(* CODESYS project filling_station_1309_Final.ecp

Project tree, tasks and I/O mapping:
  GenericDummyMasterDevice : Generic Master, WAGO, order no. None, version 1.0.0.0
  PFC200_CS_2ETH_RS : 750-8202 PFC200 2ETH RS, WAGO, order no. 0750-8202, version 1.4.1.22
    application Application
      libraries: ; Util, * (System); VisuDialogs, * (System)
      task PLC_Task (cyclic, interval t#10ms, priority 14) calls PLC_PRG
      task Visu_Task (cyclic, interval t#10ms, priority 14) calls VISU_PRG
      function CONVERT_PRESSURE_TO_LEVEL [ST]
      visualisation Visualization
      function READ_PRESSURE [ST]
      global variables GVL
      function XOR_MANUAL_AUTOMATIC_VALVE_CONTROL [ST]
      function READ_VALVE_POSITION [ST]
      function AVOID_SIMULT_VALVE_OPEN_AND_CLOSE [ST]
      program PLC_PRG [FBD]
      image pool ImagePool
      visualisation Visualization_1
      function ASSIGN_OUTPUTS [ST]
      function ACTUATOR [ST]
      function Manual_Control [FBD]
    DeviceAdapter
    Kbus : Kbus, WAGO, version 1.3.0.0
        unmapped channels: K-BUS diagnostics
      _8_DO_Generic : 075x-8DO, WAGO, order no. 075x-8DO, version 0.0.0.11
          settings: K-BUS Module slot index = 1
          output vbOpenSamsonValve : BOOL  // _OUT._OUT
          output vbCloseSamsonValve : BOOL  // _OUT._OUT
          output vbOpenDrainValveBelowWaterColumn : BOOL  // _OUT._OUT
          output vbSwitchOnPump : BOOL  // _OUT._OUT
          unmapped channels: _OUT
        DeviceAdapter
      _4_AI_0_10V_DC_s_e : 0750-0459, WAGO, order no. 0750-0459, version 0.0.0.11
          settings: K-BUS Module slot index = 2
          input  vwRawValvePosition : WORD  // _IW 1
          unmapped channels: _IW 2, _IW 3, _IW 4
        DeviceAdapter
      _2_AI_4_20mA_Diff_Measurement_Input : 0750-0492, WAGO, order no. 0750-0492, version 0.0.0.7
          settings: K-BUS Module slot index = 3
          input  vwRawPressure : WORD  // _IW 1
          unmapped channels: _IW 2
        DeviceAdapter
    MODBUS
      MODBUS : MODBUS, WAGO, order no. n/a, version 1.1.1.13
    Serial
      COM1 : COM1, WAGO, version 0.0.0.19
  e_DISPLAY_7300T_WP_10_1_1280x800_PIO1 : 0762-3003 e!DISPLAY 7300T - WP 10.1, WAGO, order no. 0762-3003, version 0.0.0.3
    DeviceAdapter
  libraries: WagoVisuIcons, 1.0.0.7 (WAGO)
  text list GlobalTextList
  5ce3da45-db07-42e7-a21c-a00fff4ed8f6|C:\Users\Alexander Wilms\Documents\Ausbildung\Hochschule Darmstadt\Master Electrical Engineering\1. Semester\Team Project\team-project\40_Implementation\hydraulics-schematic-simplified.png
  5ce3da45-db07-42e7-a21c-a00fff4ed8f6|C:\Users\Alexander Wilms\Documents\Ausbildung\Hochschule Darmstadt\Master Electrical Engineering\1. Semester\Team Project\team-project\30_Architecture\hydraulics-schematic-simplified.png
*)

// PFC200_CS_2ETH_RS/Application/GVL
VAR_GLOBAL
	vrWaterLevel:REAL;
	vrgrWaterLevel:ARRAY[1..16] OF REAL;
	vrStandardGravity:REAL:=9.81;
	viDensityWater:INT:=1000;
	vrValvePosition:REAL;
	vrValvePositionPercentage:REAL;
	vrValvePositionDesired:REAL;
	viPumpPowerPercentage:INT;
	vbManualValveControl:BOOL:=TRUE;
	vbAutomaticValveControl:BOOL:=FALSE;
	vbPreviousValveControl:STRING:='MANUAL';
	vbPreviousSamsonValveDirection:STRING:='STOP';
	vbStopSamsonValve:BOOL:=TRUE;
	vbOpenSamsonValveButton:BOOL;
	vbCloseSamsonValveButton:BOOL;
	vbOpenSamsonValveCtrl:BOOL;
	vbCloseSamsonValveCtrl:BOOL;
	vbSwitchOnPumpCtrl:BOOL:=FALSE;
	vbTrash: BOOL;
	vrController_Level_SP:REAL;
	vrController_PV:REAL;
	vbController_Manual_Mode:BOOL:=TRUE;
	vrController_Output:REAL;
	vrController_Output_reversed:REAL;
	Water_Valve_Open: BOOL;
	Water_Valve_Close: BOOL;
	PID_1: PID;
	vbOpenDrainValveBelowWaterColumnCtrl: BOOL;
END_VAR
VAR_GLOBAL RETAIN
	KP: REAL:=0.7;
	TN: REAL:=3;
	TV: REAL:=0;
END_VAR

// PFC200_CS_2ETH_RS/Application/PLC_PRG
PROGRAM PLC_PRG
VAR
	PID_0: PID;
	TRASH: BOOL;
END_VAR

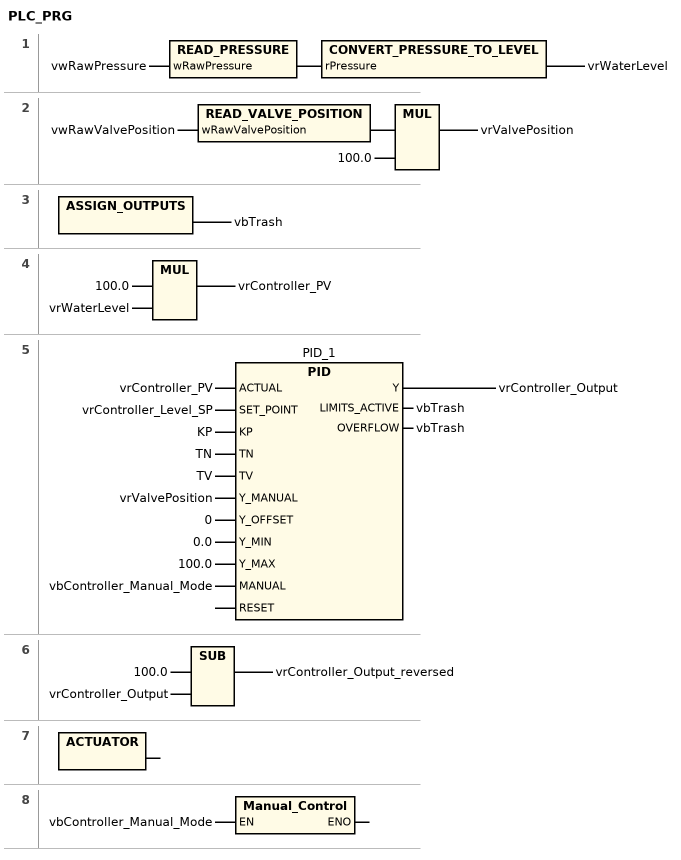
// NETWORK 1
vrWaterLevel := CONVERT_PRESSURE_TO_LEVEL(rPressure := READ_PRESSURE(wRawPressure := vwRawPressure));

// NETWORK 2
vrValvePosition := READ_VALVE_POSITION(wRawValvePosition := vwRawValvePosition) * 100.0;

// NETWORK 3
vbTrash := ASSIGN_OUTPUTS();

// NETWORK 4
vrController_PV := 100.0 * vrWaterLevel;

// NETWORK 5
PID_1(
    ACTUAL := vrController_PV,
    SET_POINT := vrController_Level_SP,
    KP := KP,
    TN := TN,
    TV := TV,
    Y_MANUAL := vrValvePosition,
    Y_OFFSET := 0,
    Y_MIN := 0.0,
    Y_MAX := 100.0,
    MANUAL := vbController_Manual_Mode,
    LIMITS_ACTIVE => vbTrash,
    OVERFLOW => vbTrash); // PID
vrController_Output := PID_1.Y;

// NETWORK 6
vrController_Output_reversed := 100.0 - vrController_Output;

// NETWORK 7
ACTUATOR();

// NETWORK 8
IF vbController_Manual_Mode THEN Manual_Control(); END_IF

END_PROGRAM

// PFC200_CS_2ETH_RS/Application/CONVERT_PRESSURE_TO_LEVEL
FUNCTION CONVERT_PRESSURE_TO_LEVEL : REAL
VAR_INPUT
	rPressure:REAL;
END_VAR
VAR
END_VAR

CONVERT_PRESSURE_TO_LEVEL := rPressure/viDensityWater/vrStandardGravity;

END_FUNCTION

// PFC200_CS_2ETH_RS/Application/READ_PRESSURE
FUNCTION READ_PRESSURE : REAL
VAR_INPUT
	wRawPressure:WORD;
END_VAR
VAR
END_VAR

READ_PRESSURE := WORD_TO_REAL((wRawPressure)*9810*2)/65535;

END_FUNCTION

// PFC200_CS_2ETH_RS/Application/READ_VALVE_POSITION
FUNCTION READ_VALVE_POSITION : REAL
VAR_INPUT
	wRawValvePosition:WORD;
END_VAR
VAR
END_VAR

IF (wRawValvePosition<3840)
	THEN 
	wRawValvePosition:= 3840;
END_IF
READ_VALVE_POSITION := WORD_TO_REAL (1)-WORD_TO_REAL(wRawValvePosition-3840)/(32764-3840);
vrValvePositionPercentage := READ_VALVE_POSITION*100;

END_FUNCTION

// PFC200_CS_2ETH_RS/Application/ASSIGN_OUTPUTS
FUNCTION ASSIGN_OUTPUTS : BOOL
VAR_INPUT
END_VAR
VAR
END_VAR

vbSwitchOnPump:=vbSwitchOnPumpCtrl;
vbOpenDrainValveBelowWaterColumn:=vbOpenDrainValveBelowWaterColumnCtrl;
vbOpenSamsonValveCtrl:=vbOpenSamsonValve;
vbCloseSamsonValveCtrl:=vbCloseSamsonValve;
ASSIGN_OUTPUTS:=TRUE;

END_FUNCTION

// PFC200_CS_2ETH_RS/Application/ACTUATOR
FUNCTION ACTUATOR : BOOL
VAR_INPUT
END_VAR
VAR
END_VAR

IF vbController_Manual_Mode=FALSE
	THEN
	vbOpenSamsonValveButton:=FALSE;
	vbCloseSamsonValveButton:=FALSE;
	
	END_IF

IF (vrController_Output_reversed - vrValvePosition) <= 3 AND (vrValvePosition - vrController_Output_reversed) <= 3 AND (vbController_Manual_Mode=FALSE)
  		THEN
	vbOpenSamsonValve:=vbOpenSamsonValve;
	vbCloseSamsonValve:=vbCloseSamsonValve;
ELSIF (vrController_Output_reversed - vrValvePosition) > 3  AND (vbController_Manual_Mode=FALSE)
	THEN
	vbOpenSamsonValve:=TRUE;
	vbCloseSamsonValve:=FALSE;
ELSIF (vbController_Manual_Mode=FALSE)
  		THEN
vbOpenSamsonValve:=FALSE;
vbCloseSamsonValve:=TRUE;
END_IF

END_FUNCTION

// PFC200_CS_2ETH_RS/Application/Manual_Control
FUNCTION Manual_Control : BOOL
VAR_INPUT
	
END_VAR
VAR
	RS_2: RS;
	RS_3: RS;
END_VAR

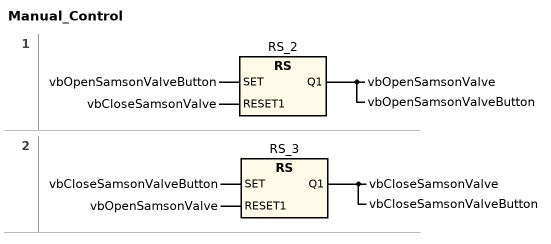
// NETWORK 1
RS_2(SET := vbOpenSamsonValveButton, RESET1 := vbCloseSamsonValve); // RS
vbOpenSamsonValve := RS_2.Q1;
vbOpenSamsonValveButton := RS_2.Q1;

// NETWORK 2
RS_3(SET := vbCloseSamsonValveButton, RESET1 := vbOpenSamsonValve); // RS
vbCloseSamsonValve := RS_3.Q1;
vbCloseSamsonValveButton := RS_3.Q1;

END_FUNCTION

// PFC200_CS_2ETH_RS/Application/XOR_MANUAL_AUTOMATIC_VALVE_CONTROL
FUNCTION XOR_MANUAL_AUTOMATIC_VALVE_CONTROL : BOOL
VAR_INPUT
END_VAR
VAR
END_VAR

IF vbAutomaticValveControl AND vbManualValveControl THEN
	IF vbPreviousValveControl = 'MANUAL' THEN
			vbAutomaticValveControl := TRUE;
			vbManualValveControl := FALSE;
			vbPreviousValveControl := 'AUTOMATIC';
	ELSIF
			vbPreviousValveControl =  'AUTOMATIC' THEN
			vbAutomaticValveControl := FALSE;
			vbManualValveControl := TRUE;
			vbPreviousValveControl := 'MANUAL';
	END_IF
END_IF

XOR_MANUAL_AUTOMATIC_VALVE_CONTROL := TRUE;

END_FUNCTION

// PFC200_CS_2ETH_RS/Application/AVOID_SIMULT_VALVE_OPEN_AND_CLOSE
FUNCTION AVOID_SIMULT_VALVE_OPEN_AND_CLOSE : BOOL
VAR_INPUT
END_VAR
VAR
END_VAR

IF vbOpenSamsonValve AND vbStopSamsonValve THEN
	IF vbPreviousSamsonValveDirection = 'OPEN' THEN
		vbOpenSamsonValve := FALSE;
		vbStopSamsonValve := TRUE;
		vbCloseSamsonValve := FALSE;
		vbPreviousSamsonValveDirection := 'STOP';
	ELSIF vbPreviousSamsonValveDirection = 'STOP' THEN
		vbOpenSamsonValve := TRUE;
		vbStopSamsonValve := FALSE;
		vbCloseSamsonValve := FALSE;
		vbPreviousSamsonValveDirection := 'OPEN';
	END_IF
ELSIF vbStopSamsonValve AND vbCloseSamsonValve THEN
	IF vbPreviousSamsonValveDirection = 'STOP' THEN
		vbOpenSamsonValve := FALSE;
		vbStopSamsonValve := FALSE;
		vbCloseSamsonValve := TRUE;
		vbPreviousSamsonValveDirection := 'CLOSE';
	ELSIF vbPreviousSamsonValveDirection = 'CLOSE' THEN
		vbOpenSamsonValve := FALSE;
		vbStopSamsonValve := TRUE;
		vbCloseSamsonValve := FALSE;
		vbPreviousSamsonValveDirection := 'STOP';
	END_IF
ELSIF vbOpenSamsonValve AND vbCloseSamsonValve THEN
	IF vbPreviousSamsonValveDirection = 'OPEN' THEN
		vbOpenSamsonValve := FALSE;
		vbStopSamsonValve := FALSE;
		vbCloseSamsonValve := TRUE;
		vbPreviousSamsonValveDirection := 'CLOSE';
	ELSIF vbPreviousSamsonValveDirection = 'CLOSE' THEN
		vbOpenSamsonValve := TRUE;
		vbStopSamsonValve := FALSE;
		vbCloseSamsonValve := FALSE;
		vbPreviousSamsonValveDirection := 'OPEN';
	END_IF
END_IF

AVOID_SIMULT_VALVE_OPEN_AND_CLOSE := TRUE;

END_FUNCTION

// PFC200_CS_2ETH_RS/Application/Visualization
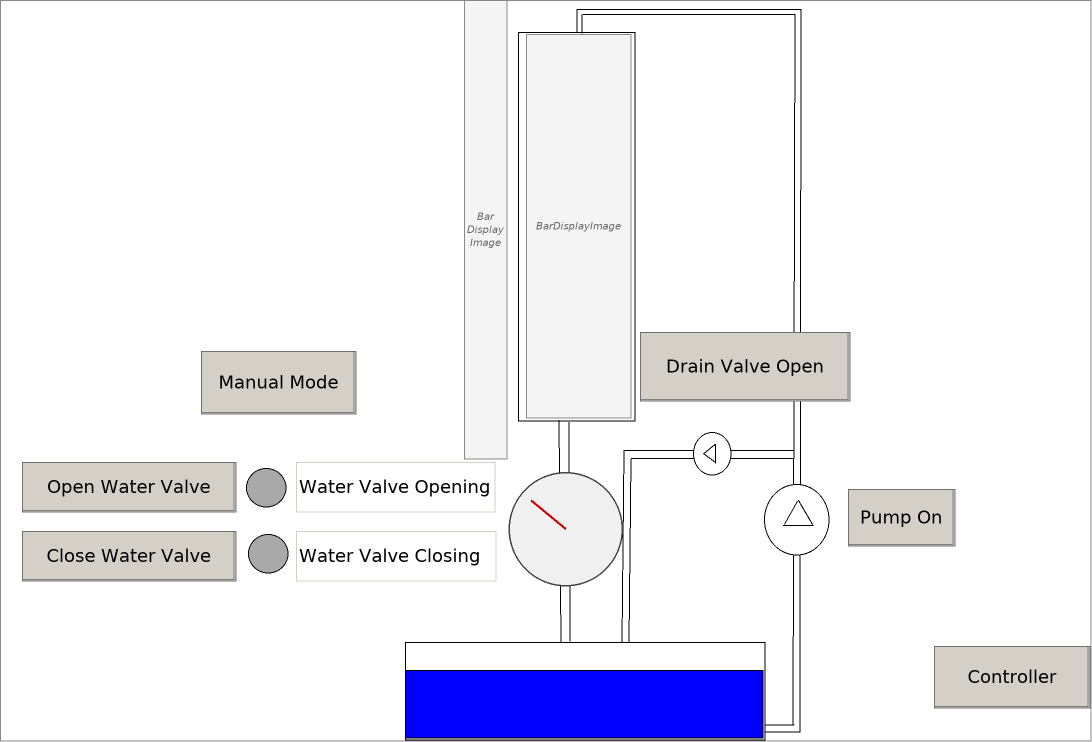
VISUALIZATION Visualization  // 1092x742
    Button (934,646 156x62), "Controller"
        OnMouseClick:  Assign=Visualization_1, Type=Assignment
    RoundedRectangle (518,32 117x389)
    BarDisplayImage (526,34 105x384), value: vrWaterLevel, style: BarDisplayImage-Gray, scale format: %.1f, scale 0..1
        p518627256: m
    Line (577,32) (577,9)
    Line (583,14) (794,14)
    Line (577,9) (801,9)
    Line (582,33) (582,14)
    Line (740,9) (740,9)
    Line (800,732) (801,9)
    Rectangle (405,642 360x98)
    Line (800,732) (765,732)
    Line (794,725) (765,725)
    Line (793,725) (795,14)
    Line (561,642) (559,420)
    Line (629,642) (631,459)
    Group (764,484 65x71), colour toggle: vbSwitchOnPumpCtrl
        Ellipse (0,0 65x71), colour toggle: vbSwitchOnPumpCtrl
        Line (34,16) (48,40)
        Line (33,17) (20,40)
        Line (19,41) (49,41)
    Button (848,489 107x57), "Pump On", colour toggle: vbSwitchOnPumpCtrl
        OnMouseClick:  ToggleVariable=vbSwitchOnPumpCtrl
    BarDisplayImage (464,0 43x459), value: vrWaterLevel, style: BarDisplayImage-Gray, scale format: %.1f, scale 0..1
        p518627256: m
    Line (570,641) (569,422)
    Line (622,642) (624,450)
    Meter360 (507,472 117x114), value: vrValvePositionPercentage, style: Meter-Meter360-Gray, scale format: %.0f, scale 0..100
        p518627256: %
    Rectangle (405,670 358x68)
    Button (640,332 210x69), "Drain Valve Open", colour toggle: vbOpenDrainValveBelowWaterColumnCtrl
        OnMouseClick:  ToggleVariable=vbOpenDrainValveBelowWaterColumnCtrl
    Ellipse (246,468 40x39), colour toggle: vbOpenSamsonValveCtrl
    Ellipse (248,534 40x39), colour toggle: vbCloseSamsonValveCtrl
    Textfield (296,462 199x50), "Water Valve Opening"
    Textfield (296,531 200x50), "Water Valve Closing"
    Button (201,351 155x63), "Manual Mode", colour toggle: vbController_Manual_Mode
        OnMouseClick:  ToggleVariable=vbController_Manual_Mode
        OnDialogClosed:  ToggleVariable=vbController_Manual_Mode
    Button (22,462 214x50), "Open Water Valve", colour toggle: vbOpenSamsonValveButton
        OnMouseClick:  ToggleVariable=vbOpenSamsonValveButton
    Button (22,531 214x50), "Close Water Valve", colour toggle: vbCloseSamsonValveButton
        OnMouseClick:  ToggleVariable=vbCloseSamsonValveButton
    Line (624,450) (794,450)
    Line (631,458) (794,458)
    Ellipse (693,432 38x43), colour toggle: vbOpenDrainValveBelowWaterColumnCtrl
    Line (703,453) (715,462)
    Line (715,444) (715,463)
    Line (704,453) (715,444)
END_VISUALIZATION

// PFC200_CS_2ETH_RS/Application/Visualization_1
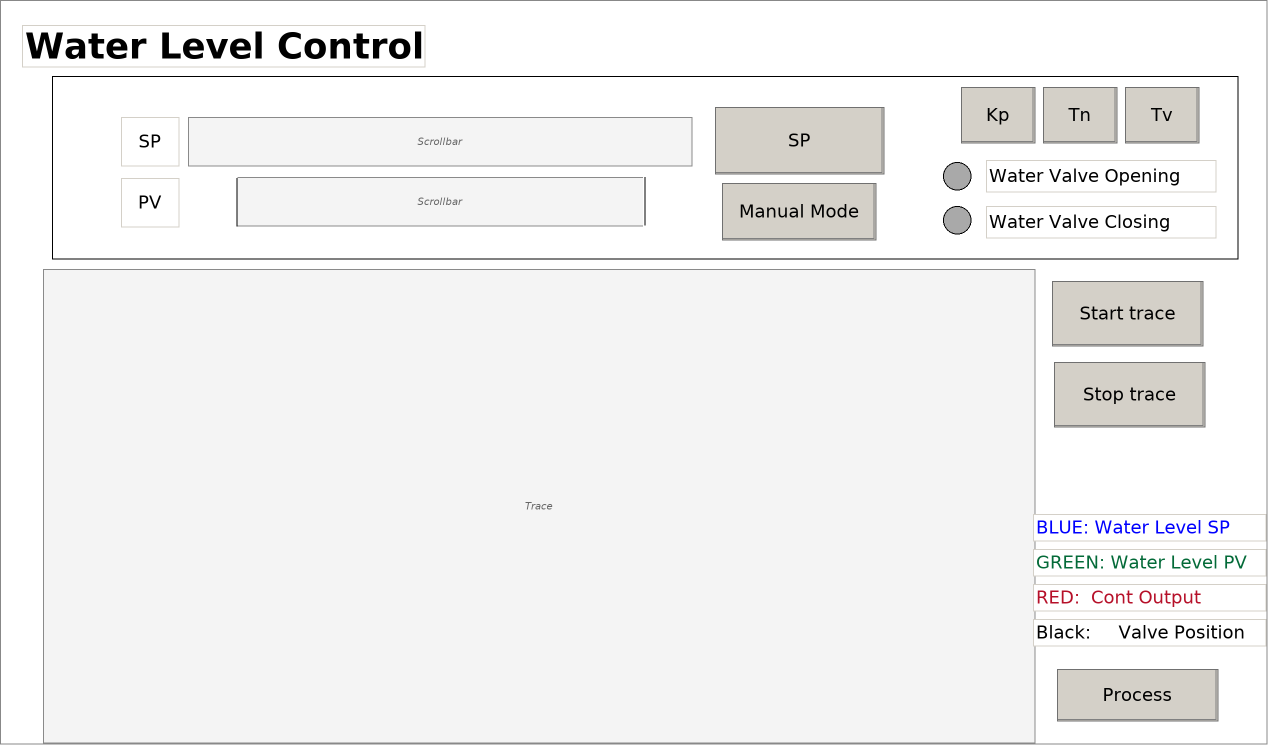
VISUALIZATION Visualization_1  // 1268x745
VAR_IN_OUT
END_VAR
VAR
	bResetTrigger : BOOL;
	bStart : BOOL;
	bStop : BOOL;
	bStore : BOOL;
	sStoreFilename : STRING;
	bRestore : BOOL;
	sRestoreFilename : STRING;
END_VAR
    RoundedRectangle (52,76 1186x183)
    Button (1057,669 161x52), "Process"
        OnMouseClick:  Assign=Visualization, Type=Assignment
    Scrollbar (188,117 504x49), text variable: vrController_Level_SP
        p1057716461: vrController_Level_SP
        p2175578022: vrController_Level_SP
    Trace (43,269 992x474)
        p3825648158: bResetTrigger
        p866368322: bStart
        p3851742229: bStop
        p2132035699: bStore
        p163910951: sStoreFilename
        p2217859334: bRestore
        p1301606187: sRestoreFilename
    Button (1052,281 151x65), "Start trace"
        toggle bStart
    Button (1054,362 151x65), "Stop trace"
        toggle bStop
    Textfield (1033,514 233x27), "BLUE: Water Level SP"
    Textfield (1033,549 233x27), "GREEN: Water Level PV"
    Textfield (1033,584 233x27), "RED: Cont Output"
    Textfield (1033,619 233x27), "Black: Valve Position"
    Button (722,183 154x57), "Manual Mode", colour toggle: vbController_Manual_Mode
        OnMouseClick:  ToggleVariable=vbController_Manual_Mode
        OnDialogClosed:  ToggleVariable=vbController_Manual_Mode
    Ellipse (943,162 28x28), colour toggle: vbOpenSamsonValveCtrl
    Ellipse (943,206 28x28), colour toggle: vbCloseSamsonValveCtrl
    Textfield (986,160 230x32), "Water Valve Opening"
    Textfield (986,206 230x32), "Water Valve Closing"
    Textfield (121,117 58x49), "SP"
    Textfield (121,178 58x49), "PV"
    Scrollbar (188,177 504x49), text variable: vrController_Level_SP
        p1057716461: vrController_PV
        p2175578022: vrController_Level_SP
    Textfield (22,25 403x42), "Water Level Control"
    Button (715,107 169x67), "SP"
        OnMouseClick: write vrController_Level_SP via Default, min 0, max 100, format %.f
    Button (1043,87 74x56), "Tn"
        OnMouseClick: write TN via Default, min 0.0, max 30.0, format %.1f
    Button (1125,87 74x56), "Tv"
        OnMouseClick: write TV via Default, min 0.0, max 30.0, format %.1f
    Button (961,87 74x56), "Kp"
        OnMouseClick: write KP via Default, min 0.0, max 2.0, format %.1f
    RoundedRectangle (185,175 52x52)
    RoundedRectangle (643,175 52x52)
    Line (237,226) (237,178)
    Line (645,225) (645,177)
END_VISUALIZATION
